Fanuc KAREL source: ka00119.KL

-- PROVISIONAL review KL for V770-1; original PC SHA256 4570d9affb2617a90d9db5dad97a2f53e660480cf6002340ee56e6e0c41fda3a
-- Incomplete behavior may be omitted. Consult companion uncertainty JSON. Do not deploy.
PROGRAM KA00119
%NOLOCKGROUP
-- UNRESOLVED_DECL SRC type=00001c
-- UNRESOLVED_DECL DST type=002018
BEGIN
  -- UNRESOLVED_PC offsets 5-15; opcodes 9D,22,A5
  -- UNRESOLVED_PC offsets 20-35; opcodes 21,22,9D,33,B2
  -- UNRESOLVED_PC offsets 40-44; opcodes 7F
END KA00119
